// TIA Portal V20 export
TYPE "type_emRelations_em4_SoftCam"
// stored: Access Published, Namespace Unit1
   STRUCT
      anodeMainPnP1AxisX : Struct
         reelCutConveyerPos : "LER_typeSoftcamControlNodes";
         alignTablePos : "LER_typeSoftcamControlNodes";
         Pos2 { S7_SetPoint := 'True'} : "LER_typeSoftcamControlNodes";
         Pos3 { S7_SetPoint := 'True'} : "LER_typeSoftcamControlNodes";
         Pos4 { S7_SetPoint := 'True'} : "LER_typeSoftcamControlNodes";
         Pos5 { S7_SetPoint := 'True'} : "LER_typeSoftcamControlNodes";
         Pos6 { S7_SetPoint := 'True'} : "LER_typeSoftcamControlNodes";
         Pos7 { S7_SetPoint := 'True'} : "LER_typeSoftcamControlNodes";
         Pos8 { S7_SetPoint := 'True'} : "LER_typeSoftcamControlNodes";
         Pos9 { S7_SetPoint := 'True'} : "LER_typeSoftcamControlNodes";
         Pos10 { S7_SetPoint := 'True'} : "LER_typeSoftcamControlNodes";
         Pos11 { S7_SetPoint := 'True'} : "LER_typeSoftcamControlNodes";
         Pos12 { S7_SetPoint := 'True'} : "LER_typeSoftcamControlNodes";
         Pos13 { S7_SetPoint := 'True'} : "LER_typeSoftcamControlNodes";
         Pos14 { S7_SetPoint := 'True'} : "LER_typeSoftcamControlNodes";
         Pos15 { S7_SetPoint := 'True'} : "LER_typeSoftcamControlNodes";
      END_STRUCT;
      anodeMainPnP2AxisX : Struct
         alignTablePos : "LER_typeSoftcamControlNodes";
         stackTablePos : "LER_typeSoftcamControlNodes";
         Pos2 { S7_SetPoint := 'True'} : "LER_typeSoftcamControlNodes";
         Pos3 { S7_SetPoint := 'True'} : "LER_typeSoftcamControlNodes";
         Pos4 { S7_SetPoint := 'True'} : "LER_typeSoftcamControlNodes";
         Pos5 { S7_SetPoint := 'True'} : "LER_typeSoftcamControlNodes";
         Pos6 { S7_SetPoint := 'True'} : "LER_typeSoftcamControlNodes";
         Pos7 { S7_SetPoint := 'True'} : "LER_typeSoftcamControlNodes";
         Pos8 { S7_SetPoint := 'True'} : "LER_typeSoftcamControlNodes";
         Pos9 { S7_SetPoint := 'True'} : "LER_typeSoftcamControlNodes";
         Pos10 { S7_SetPoint := 'True'} : "LER_typeSoftcamControlNodes";
         Pos11 { S7_SetPoint := 'True'} : "LER_typeSoftcamControlNodes";
         Pos12 { S7_SetPoint := 'True'} : "LER_typeSoftcamControlNodes";
         Pos13 { S7_SetPoint := 'True'} : "LER_typeSoftcamControlNodes";
         Pos14 { S7_SetPoint := 'True'} : "LER_typeSoftcamControlNodes";
         Pos15 { S7_SetPoint := 'True'} : "LER_typeSoftcamControlNodes";
      END_STRUCT;
      anodeMainPnP1AxisY : Struct
         waitPos : "LER_typeSoftcamControlNodes";
         Pos1 { S7_SetPoint := 'True'} : "LER_typeSoftcamControlNodes";
         Pos2 { S7_SetPoint := 'True'} : "LER_typeSoftcamControlNodes";
         Pos3 { S7_SetPoint := 'True'} : "LER_typeSoftcamControlNodes";
         Pos4 { S7_SetPoint := 'True'} : "LER_typeSoftcamControlNodes";
         Pos5 { S7_SetPoint := 'True'} : "LER_typeSoftcamControlNodes";
         Pos6 { S7_SetPoint := 'True'} : "LER_typeSoftcamControlNodes";
         Pos7 { S7_SetPoint := 'True'} : "LER_typeSoftcamControlNodes";
         Pos8 { S7_SetPoint := 'True'} : "LER_typeSoftcamControlNodes";
         Pos9 { S7_SetPoint := 'True'} : "LER_typeSoftcamControlNodes";
         Pos10 { S7_SetPoint := 'True'} : "LER_typeSoftcamControlNodes";
         Pos11 { S7_SetPoint := 'True'} : "LER_typeSoftcamControlNodes";
         Pos12 { S7_SetPoint := 'True'} : "LER_typeSoftcamControlNodes";
         Pos13 { S7_SetPoint := 'True'} : "LER_typeSoftcamControlNodes";
         Pos14 { S7_SetPoint := 'True'} : "LER_typeSoftcamControlNodes";
         Pos15 { S7_SetPoint := 'True'} : "LER_typeSoftcamControlNodes";
      END_STRUCT;
      anodeMainPnP1AxisZ : Struct
         upPos : "LER_typeSoftcamControlNodes";
         reelCutConveyerDownPos : "LER_typeSoftcamControlNodes";
         ailgnTableDownPos : "LER_typeSoftcamControlNodes";
         avoidPos : "LER_typeSoftcamControlNodes";
         Pos4 { S7_SetPoint := 'True'} : "LER_typeSoftcamControlNodes";
         Pos5 { S7_SetPoint := 'True'} : "LER_typeSoftcamControlNodes";
         Pos6 { S7_SetPoint := 'True'} : "LER_typeSoftcamControlNodes";
         Pos7 { S7_SetPoint := 'True'} : "LER_typeSoftcamControlNodes";
         Pos8 { S7_SetPoint := 'True'} : "LER_typeSoftcamControlNodes";
         Pos9 { S7_SetPoint := 'True'} : "LER_typeSoftcamControlNodes";
         Pos10 { S7_SetPoint := 'True'} : "LER_typeSoftcamControlNodes";
         Pos11 { S7_SetPoint := 'True'} : "LER_typeSoftcamControlNodes";
         Pos12 { S7_SetPoint := 'True'} : "LER_typeSoftcamControlNodes";
         Pos13 { S7_SetPoint := 'True'} : "LER_typeSoftcamControlNodes";
         Pos14 { S7_SetPoint := 'True'} : "LER_typeSoftcamControlNodes";
         Pos15 { S7_SetPoint := 'True'} : "LER_typeSoftcamControlNodes";
      END_STRUCT;
      anodeMainPnP2AxisZ : Struct
         upPos : "LER_typeSoftcamControlNodes";
         ailgnTableDownPos : "LER_typeSoftcamControlNodes";
         stackTableDownPos : "LER_typeSoftcamControlNodes";
         avoidPos : "LER_typeSoftcamControlNodes";
         Pos4 { S7_SetPoint := 'True'} : "LER_typeSoftcamControlNodes";
         Pos5 { S7_SetPoint := 'True'} : "LER_typeSoftcamControlNodes";
         Pos6 { S7_SetPoint := 'True'} : "LER_typeSoftcamControlNodes";
         Pos7 { S7_SetPoint := 'True'} : "LER_typeSoftcamControlNodes";
         Pos8 { S7_SetPoint := 'True'} : "LER_typeSoftcamControlNodes";
         Pos9 { S7_SetPoint := 'True'} : "LER_typeSoftcamControlNodes";
         Pos10 { S7_SetPoint := 'True'} : "LER_typeSoftcamControlNodes";
         Pos11 { S7_SetPoint := 'True'} : "LER_typeSoftcamControlNodes";
         Pos12 { S7_SetPoint := 'True'} : "LER_typeSoftcamControlNodes";
         Pos13 { S7_SetPoint := 'True'} : "LER_typeSoftcamControlNodes";
         Pos14 { S7_SetPoint := 'True'} : "LER_typeSoftcamControlNodes";
         Pos15 { S7_SetPoint := 'True'} : "LER_typeSoftcamControlNodes";
      END_STRUCT;
      anodeAlignTableAxisX : Struct
         waitPos : "LER_typeSoftcamControlNodes";
         adjustPos : "LER_typeSoftcamControlNodes";
         Pos2 { S7_SetPoint := 'True'} : "LER_typeSoftcamControlNodes";
         Pos3 { S7_SetPoint := 'True'} : "LER_typeSoftcamControlNodes";
         Pos4 { S7_SetPoint := 'True'} : "LER_typeSoftcamControlNodes";
         Pos5 { S7_SetPoint := 'True'} : "LER_typeSoftcamControlNodes";
         Pos6 { S7_SetPoint := 'True'} : "LER_typeSoftcamControlNodes";
         Pos7 { S7_SetPoint := 'True'} : "LER_typeSoftcamControlNodes";
         Pos8 { S7_SetPoint := 'True'} : "LER_typeSoftcamControlNodes";
         Pos9 { S7_SetPoint := 'True'} : "LER_typeSoftcamControlNodes";
         Pos10 { S7_SetPoint := 'True'} : "LER_typeSoftcamControlNodes";
         Pos11 { S7_SetPoint := 'True'} : "LER_typeSoftcamControlNodes";
         Pos12 { S7_SetPoint := 'True'} : "LER_typeSoftcamControlNodes";
         Pos13 { S7_SetPoint := 'True'} : "LER_typeSoftcamControlNodes";
         Pos14 { S7_SetPoint := 'True'} : "LER_typeSoftcamControlNodes";
         Pos15 { S7_SetPoint := 'True'} : "LER_typeSoftcamControlNodes";
      END_STRUCT;
      anodeAlignTableAxisY1 : Struct
         waitPos : "LER_typeSoftcamControlNodes";
         adjustPos : "LER_typeSoftcamControlNodes";
         Pos2 { S7_SetPoint := 'True'} : "LER_typeSoftcamControlNodes";
         Pos3 { S7_SetPoint := 'True'} : "LER_typeSoftcamControlNodes";
         Pos4 { S7_SetPoint := 'True'} : "LER_typeSoftcamControlNodes";
         Pos5 { S7_SetPoint := 'True'} : "LER_typeSoftcamControlNodes";
         Pos6 { S7_SetPoint := 'True'} : "LER_typeSoftcamControlNodes";
         Pos7 { S7_SetPoint := 'True'} : "LER_typeSoftcamControlNodes";
         Pos8 { S7_SetPoint := 'True'} : "LER_typeSoftcamControlNodes";
         Pos9 { S7_SetPoint := 'True'} : "LER_typeSoftcamControlNodes";
         Pos10 { S7_SetPoint := 'True'} : "LER_typeSoftcamControlNodes";
         Pos11 { S7_SetPoint := 'True'} : "LER_typeSoftcamControlNodes";
         Pos12 { S7_SetPoint := 'True'} : "LER_typeSoftcamControlNodes";
         Pos13 { S7_SetPoint := 'True'} : "LER_typeSoftcamControlNodes";
         Pos14 { S7_SetPoint := 'True'} : "LER_typeSoftcamControlNodes";
         Pos15 { S7_SetPoint := 'True'} : "LER_typeSoftcamControlNodes";
      END_STRUCT;
      anodeAlignTableAxisY2 : Struct
         waitPos : "LER_typeSoftcamControlNodes";
         adjustPos : "LER_typeSoftcamControlNodes";
         Pos2 { S7_SetPoint := 'True'} : "LER_typeSoftcamControlNodes";
         Pos3 { S7_SetPoint := 'True'} : "LER_typeSoftcamControlNodes";
         Pos4 { S7_SetPoint := 'True'} : "LER_typeSoftcamControlNodes";
         Pos5 { S7_SetPoint := 'True'} : "LER_typeSoftcamControlNodes";
         Pos6 { S7_SetPoint := 'True'} : "LER_typeSoftcamControlNodes";
         Pos7 { S7_SetPoint := 'True'} : "LER_typeSoftcamControlNodes";
         Pos8 { S7_SetPoint := 'True'} : "LER_typeSoftcamControlNodes";
         Pos9 { S7_SetPoint := 'True'} : "LER_typeSoftcamControlNodes";
         Pos10 { S7_SetPoint := 'True'} : "LER_typeSoftcamControlNodes";
         Pos11 { S7_SetPoint := 'True'} : "LER_typeSoftcamControlNodes";
         Pos12 { S7_SetPoint := 'True'} : "LER_typeSoftcamControlNodes";
         Pos13 { S7_SetPoint := 'True'} : "LER_typeSoftcamControlNodes";
         Pos14 { S7_SetPoint := 'True'} : "LER_typeSoftcamControlNodes";
         Pos15 { S7_SetPoint := 'True'} : "LER_typeSoftcamControlNodes";
      END_STRUCT;
   END_STRUCT;
END_TYPE
